# EPICS substitutions: indfurnSup/indfurn_pid.substitutions
file indfurn_pid.template {

pattern {PORT, P, CTRL}
{"\$(PORT)", "\$(P)", "P"}
{"\$(PORT)", "\$(P)", "I"}
{"\$(PORT)", "\$(P)", "D"}
}
